(* PLC project cmd_on_off_pump, Dassault Systèmes ControlBuild 2024x *)
(* stored: creationDateTime 2023-10-03T11:13:36-01:00 *)

FUNCTION_BLOCK actuator
  VAR_INPUT
    autoMode : BOOL := false;
    manualMode : BOOL := false;
  END_VAR
  VAR_INPUT
    autoCmd : BOOL := false;
  END_VAR
  VAR_INPUT
    onPB : BOOL := false;
    offPB : BOOL := false;
  END_VAR
  VAR_INPUT
    generalFault : BOOL := false;
  END_VAR
  VAR_OUTPUT
    cmd : BOOL := false;
  END_VAR

(* LD diagram, written out as Structured Text *)
1:
cmd := (autoMode AND autoCmd OR manualMode AND (onPB OR cmd) AND NOT offPB) AND NOT generalFault;
END_FUNCTION_BLOCK

FUNCTION_BLOCK faults
  VAR_INPUT
    cmd : BOOL := false;
  END_VAR
  VAR_INPUT
    thermalFB : BOOL := false;
    onFB : BOOL := false;
  END_VAR
  VAR_INPUT
    acknowledgePB : BOOL := false;
  END_VAR
  VAR_OUTPUT
    generalFault : BOOL := false;
  END_VAR
  VAR
    thermalFault : BOOL := false;
    onFBFault : BOOL := false;
  END_VAR

(* LD diagram, written out as Structured Text *)
1:
IF acknowledgePB THEN thermalFault := FALSE; END_IF;
IF acknowledgePB THEN onFBFault := FALSE; END_IF;
IF acknowledgePB THEN generalFault := FALSE; END_IF;
2:
TON_FB(IN := cmd, PT := T#0h0m2s0ms);
IF TON_FB.Q0 AND NOT onFB THEN onFBFault := TRUE; END_IF;
3:
IF NOT thermalFB THEN thermalFault := TRUE; END_IF;
4:
IF onFBFault OR thermalFault THEN generalFault := TRUE; END_IF;
END_FUNCTION_BLOCK

(* Command of an on/off pump with fault detection *)
PROGRAM cmd_equipment_library.cmd_on_off_pump
  VAR_INPUT
    autoMode : BOOL := false;
    manualMode : BOOL := false;
  END_VAR
  VAR_INPUT
    autoCmd : BOOL := false;
  END_VAR
  VAR_INPUT
    thermalFB : BOOL := false;
    onFB : BOOL := false;
  END_VAR
  VAR_INPUT
    onPB : BOOL := false;
    offPB : BOOL := false;
  END_VAR
  VAR_INPUT
    acknowledgePB : BOOL := false;
  END_VAR
  VAR_OUTPUT
    cmd : BOOL := false;
  END_VAR
  VAR_OUTPUT
    generalFault : BOOL := false;
  END_VAR

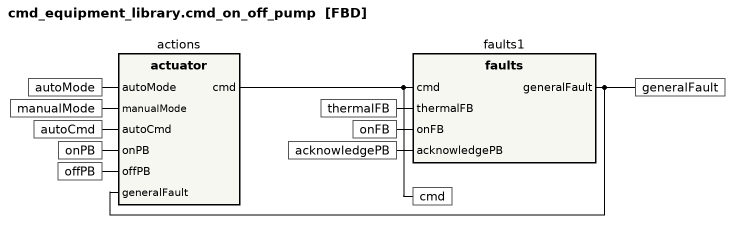
(* FBD diagram, written out as Structured Text *)
faults1(cmd := actions.cmd, thermalFB := thermalFB, onFB := onFB, acknowledgePB := acknowledgePB);
actions(autoMode := autoMode, manualMode := manualMode, autoCmd := autoCmd, onPB := onPB, offPB := offPB, generalFault := faults1.generalFault);
cmd := actions.cmd;
generalFault := faults1.generalFault;
END_PROGRAM
